Staubli VAL3: Control_BottomS.pgx

public program Control_BottomS(string x_sBottomList)
  local string l_sBottomList[8]
  local bool l_bRes
begin
      //说明：
  //函数功能：对功能键进行说明
  //x_sBottomList 功能键说明，通过字符串来实现
  //字符串以,作为分隔符



  call Str_SplitComma(l_bRes,x_sBottomList,l_sBottomList)
  if !l_bRes
    return
  endIf

call Control_Bottom(l_sBottomList)

end
